Staubli VAL3: main.pgx

public program main()
  local bool l_bSave
begin
  // INIT
  call onStart()
  // LOOP UNTIL nKey=255
  do
    call refresh()
    nKey=getKey()
    call use:listevent(nKey,nIndex,sEvent)
    nView=use:nView
    if nIndex>=0
      switch nKey
        case 259
          // TAB
          bLarge=!bLarge
          call use:setView(bLarge)
        break
        case 271
          // RESET ALL
          call onF1Event()
        break
        case 272
          // edit traj
          call onF2Event()
        break
        case 273
          call onF3Event()
        break
        case 274
          call onF4Event()
        break
        case 275
        break
        case 276
          // back
          call onF6Event(sPalletName[nIndex])
        break
        case 277
          // next
          call onF7Event(sPalletName[nIndex])
        break
        case 278
          // reset
          call onF8Event(sPalletName[nIndex])
        break
        case 270
          call onEnterEvent(sPalletName[nIndex])
        break
      endSwitch
    endIf
    // release
    delay(0)
  until nKey==255
  // on Exit
  call onExit()
end
